// TIA Portal V16 program export: 1 tag tables, 0 data types, 1 data blocks, 5 code blocks (in call order from the OBs), 0 instance data blocks

VAR_GLOBAL   // PLC tag table "Default tag table"
   inp_1_tia_da_degisti AT %M0.0 : Bool;
   out_1_degistirildi AT %M0.1 : Bool;
END_VAR

DATA_BLOCK "Data_block_1"   // DB1
{ S7_Optimized_Access := 'TRUE' }
VERSION : 0.1
// stored: AutoNumber true, DBAccessibleFromOPCUA true, IsOnlyStoredInLoadMemory false, IsRetainMemResEnabled false, IsWriteProtectedInAS false, MemoryReserve 100
   VAR
      ex : Bool;
      ex_1 : Bool;
      ex_2 : Bool;
      ex_3 : Bool;
      ex_4 : Bool;
      ex_5 : Bool;
      ex_6 : Bool;
      ex_7 : Bool;
      ex_8 : Bool;
      ex_9 : Bool;
      new : Bool;
      new_1 : Bool;
      new_2 : Bool;
   END_VAR
BEGIN
END_DATA_BLOCK

ORGANIZATION_BLOCK "Main"   // OB1, LAD, ProgramCycle
TITLE = "Main Program Sweep (Cycle)"
{ S7_Optimized_Access := 'TRUE' }
VERSION : 0.1
// stored: AutoNumber true, IsIECCheckEnabled false, SetENOAutomatically false
   VAR_INPUT
      Initial_Call : Bool;   // Initial call of this OB
      Remanence : Bool;   // =True, if remanent data are available
   END_VAR
   VAR_TEMP
      deneme_123 : Bool;
      deneme_2 : Bool;
   END_VAR
BEGIN

REGION Network 1: yorum111
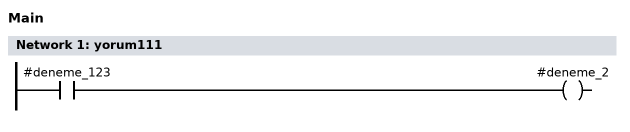
   RUNG wire#powerrail
      Contact( #deneme_123 )
      Coil( #deneme_2 )
   END_RUNG
   // the same network as SCL:
   #deneme_2 := #deneme_123;
END_REGION
END_ORGANIZATION_BLOCK

FUNCTION "Block_1" : Void   // FC2, LAD
{ S7_Optimized_Access := 'TRUE' }
VERSION : 0.1
// stored: AutoNumber true, IsIECCheckEnabled false, SetENOAutomatically false, UDAEnableTagReadback false
BEGIN
END_FUNCTION

FUNCTION "analog_output_scale" : Void   // FC1, LAD
{ S7_Optimized_Access := 'TRUE' }
VERSION : 0.1
// stored: AutoNumber true, IsIECCheckEnabled false, SetENOAutomatically false, UDAEnableTagReadback false
BEGIN

REGION Network 1
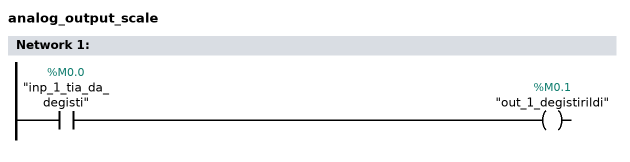
   RUNG wire#powerrail
      Contact( "inp_1_tia_da_degisti" )
      Coil( "out_1_degistirildi" )
   END_RUNG
   // the same network as SCL:
   "out_1_degistirildi" := "inp_1_tia_da_degisti";
END_REGION
END_FUNCTION

FUNCTION_BLOCK "FB548.Divert.Sorter.Chute"   // FB542, LAD
{ S7_Optimized_Access := 'TRUE' }
VERSION : 0.1
// stored: AutoNumber false, IsIECCheckEnabled false, IsRetainMemResEnabled false, MemoryReserve 100, SetENOAutomatically false, UDAEnableTagReadback false
   VAR_INPUT
      Acil_Yok : Bool;
      Sorter_Calisiyor : Bool;
      Sağ_Chute_Sorted_Sensoru : Bool;
      Sol_Chute_Sorted_Sensoru : Bool;
      "Sağ_Chute_Aktif / Pasif" : Bool;   // 1 = Aktif , 0 = Pasif
      "Sol_Chute_Aktif / Pasif" : Bool;   // 1 = Aktif , 0 = Pasif
      Chute_Rulo_Hatası : Bool;
      Divert_Sürücü_Hatası : Bool;
      Pozisyon_Olcme_Aktif : Bool;
      Sağ_Çıkış_Target { ExternalAccessible := 'False'; ExternalVisible := 'False'; ExternalWritable := 'False'} : Int;
      Sol_Çıkış_Target { ExternalAccessible := 'False'; ExternalVisible := 'False'; ExternalWritable := 'False'} : Int;
      CN_NO : Int;
      "Aktüel Encoder Değeri" : LReal;
      Birinci_Divert_Min : LReal;
      Birinci_Divert_Max : LReal;
      İkinci_Divert_Min : LReal;
      İkinci_Divert_Max : LReal;
      Max_Kutu_Adedi { ExternalAccessible := 'False'; ExternalVisible := 'False'; ExternalWritable := 'False'} : Int;
   END_VAR
   VAR_OUTPUT
      "1_sol_Divert_Çalıştır" : Bool;
      "2_sol_Divert_Çalıştır" : Bool;
      "1_sağ_Divert_Çalıştır" : Bool;
      "2_sağ_Divert_Çalıştır" : Bool;
      "Sort Hatası" : Bool;
   END_VAR
   VAR
      Sort_Aktif_AUX : Array[1..10] of Bool;
      Sort_Aktif_PTrig : Array[1..10] of Bool;
      TOF_TIME : Array[1..10] of TOF_TIME;
      TON_TIME { S7_SetPoint := 'True'} : Array[1..10] of TON_TIME;
      Sort_Aktif1 : Bool;
      Sort_Aktif2 : Bool;
      Sort_Aktif1_Sağ : Bool;
      Sort_Aktif2_Sağ : Bool;
      Sağ_Sort_Pasif : Bool;
      Sol_Sort_Pasif : Bool;
      Ikinci_Servo_Baslama : Time;
      Divert_Durdur : Bool;
      Sort_Aktif_1 { ExternalAccessible := 'False'; ExternalVisible := 'False'; ExternalWritable := 'False'} : Array[1..10] of Bool;
      Sort_Aktif_2 { ExternalAccessible := 'False'; ExternalVisible := 'False'; ExternalWritable := 'False'} : Array[1..10] of Bool;
      Sort_Aktif_1_Sağ : Array[1..10] of Bool;
      Sort_Aktif_2_Sağ : Array[1..10] of Bool;
      Sort_Ilk_Pozisyon { ExternalAccessible := 'False'; ExternalVisible := 'False'; ExternalWritable := 'False'} : Array[1..10] of LReal;
      Sort_Ön_Pozisyon { ExternalAccessible := 'False'; ExternalVisible := 'False'; ExternalWritable := 'False'} : Array[1..10] of LReal;
      Sort_Aktif_Boy { ExternalAccessible := 'False'; ExternalVisible := 'False'; ExternalWritable := 'False'} : Array[1..10] of LReal;
      SortKutuNo : Int;
   END_VAR
   VAR_TEMP
      "On/Off" : Bool;
      j : Int;
      Ekstra_Uzunluk : LReal;
   END_VAR
   VAR_TEMP   // added for the SCL form of the ladder/FBD networks
      _w1 : Bool;
      _w2 : Bool;
      _w3 : Bool;
      _w4 : Bool;
   END_VAR
BEGIN

REGION Network 1: On / Off
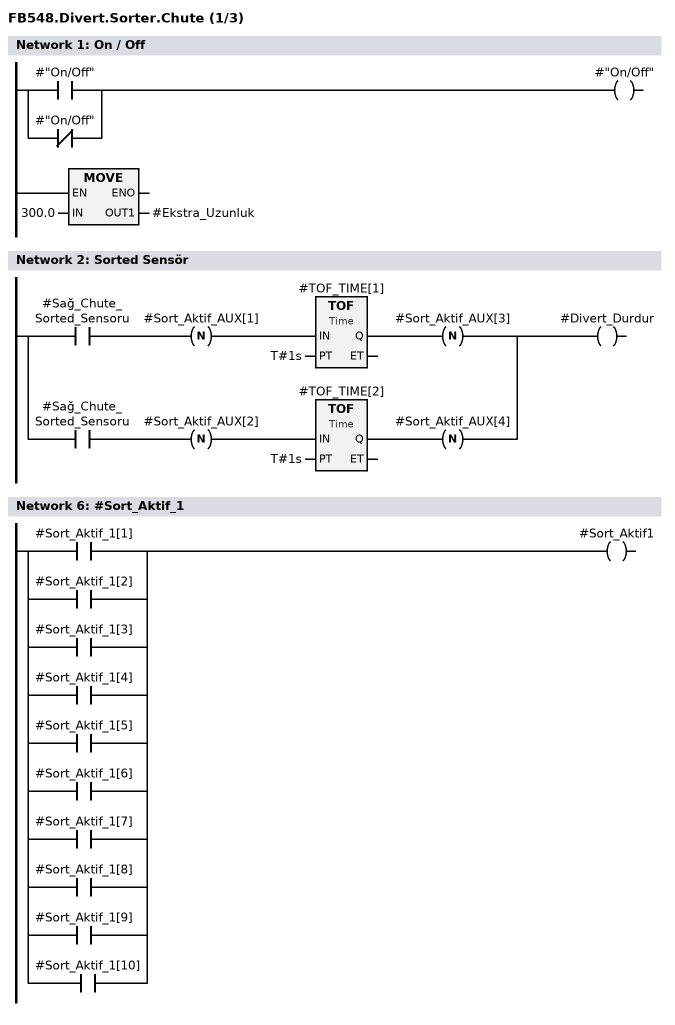
   RUNG wire#powerrail
      Contact( #"On/Off" )
      wire#w1
      Coil( #"On/Off" )
   END_RUNG
   RUNG wire#powerrail
      I_Contact( #"On/Off" )
   END_RUNG wire#w1
   RUNG wire#powerrail
      Move(in := 300.0, out1 => #Ekstra_Uzunluk)
   END_RUNG
   // the same network as SCL:
   #"On/Off" := #"On/Off" OR NOT #"On/Off";
   #Ekstra_Uzunluk := 300.0;
END_REGION

REGION Network 2: Sorted Sensör
   RUNG wire#powerrail
      Contact( #Sağ_Chute_Sorted_Sensoru )
      N_Trig( #Sort_Aktif_AUX[1] )
      { S7_Templates := "time_type := Time" } #TOF_TIME[1].TOF(pt := T#1s, et =>)
      N_Trig( #Sort_Aktif_AUX[3] )
      wire#w1
      Coil( #Divert_Durdur )
   END_RUNG
   RUNG wire#powerrail
      Contact( #Sağ_Chute_Sorted_Sensoru )
      N_Trig( #Sort_Aktif_AUX[2] )
      { S7_Templates := "time_type := Time" } #TOF_TIME[2].TOF(pt := T#1s, et =>)
      N_Trig( #Sort_Aktif_AUX[4] )
   END_RUNG wire#w1
   // the same network as SCL:
   #_w1 := NOT #Sağ_Chute_Sorted_Sensoru AND #Sort_Aktif_AUX[1];   // falling edge
   #Sort_Aktif_AUX[1] := #Sağ_Chute_Sorted_Sensoru;
   #TOF_TIME[1].TOF(IN := #_w1, PT := T#1s);
   #_w2 := NOT #TOF_TIME[1].Q AND #Sort_Aktif_AUX[3];   // falling edge
   #Sort_Aktif_AUX[3] := #TOF_TIME[1].Q;
   #_w3 := NOT #Sağ_Chute_Sorted_Sensoru AND #Sort_Aktif_AUX[2];   // falling edge
   #Sort_Aktif_AUX[2] := #Sağ_Chute_Sorted_Sensoru;
   #TOF_TIME[2].TOF(IN := #_w3, PT := T#1s);
   #_w4 := NOT #TOF_TIME[2].Q AND #Sort_Aktif_AUX[4];   // falling edge
   #Sort_Aktif_AUX[4] := #TOF_TIME[2].Q;
   #Divert_Durdur := #_w2 OR #_w4;
END_REGION

REGION Network 3 (SCL): Kutu Ön Arka Pozisyon Hesap
   // IF #Sensör.Sensor_N_Trig THEN
   //     #Sort_Ilk_Pozisyon["DB530_Kutu".CN_NO_Anlık_Kutu_Sayısı[#CN_NO]] := #"Aktüel Encoder Değeri";
   // END_IF;
   // FOR #j := 1 TO #Max_Kutu_Adedi BY 1 DO
   //     IF "DB530_Kutu".CN_NO[#CN_NO].Kutu_No[#j].VARMI = TRUE THEN
   //         #Sort_Ön_Pozisyon[#j] := #"Aktüel Encoder Değeri" - #Sort_Ilk_Pozisyon[#j];
   //     END_IF;
   // END_FOR;
END_REGION

REGION Network 4 (SCL): Sol Sort Aktif Kararı
   IF #Pozisyon_Olcme_Aktif = 0
       // AND #Sorter_Calisiyor = TRUE
       // AND #"Sol_Chute_Aktif / Pasif"
   THEN
       FOR #j := 1 TO #Max_Kutu_Adedi BY 1 DO
           IF "DB530_Kutu".CN_NO[#CN_NO].Kutu_No[#j].VARMI THEN

               IF #"Sol_Chute_Aktif / Pasif" = 1
                   AND #Chute_Rulo_Hatası = 0
                   AND #Divert_Sürücü_Hatası = 0
                   // AND #Sol_Sort_Pasif = 0
                   AND #Acil_Yok = 1
                   AND "DB530_Kutu".CN_NO[#CN_NO].Kutu_No[#j].Posizyon >= #Birinci_Divert_Min
                   AND "DB530_Kutu".CN_NO[#CN_NO].Kutu_No[#j].Posizyon <= #Birinci_Divert_Min + "DB530_Kutu".CN_NO[#CN_NO].Kutu_No[#j].Uzunluk + #Ekstra_Uzunluk
                   AND "DB530_Kutu".CN_NO[#CN_NO].Kutu_No[#j].Target = #Sol_Çıkış_Target
                   // AND "DB530_Kutu".CN_NO[#CN_NO].Kutu_No[#j].Sort_Aktifleştirildi = FALSE
               THEN
                   #Sort_Aktif_1[#j] := TRUE;
               ELSE

                   IF #j< #Max_Kutu_Adedi THEN
                       IF ("DB530_Kutu".CN_NO[#CN_NO].Kutu_No[#j + 1].VARMI AND "DB530_Kutu".CN_NO[#CN_NO].Kutu_No[#j + 1].Target = #Sol_Çıkış_Target)
                           OR ("DB530_Kutu".CN_NO[#CN_NO].Kutu_No[#j].VARMI AND "DB530_Kutu".CN_NO[#CN_NO].Kutu_No[#j].Target = #Sol_Çıkış_Target) THEN

                           #Sort_Aktif_1[#j] := TRUE;

                       ELSE
                           #Sort_Aktif_1[#j] := FALSE;
                       END_IF;

                   END_IF;

               END_IF;

               IF #"Sol_Chute_Aktif / Pasif" = 1
                   AND #Chute_Rulo_Hatası = 0
                   AND #Divert_Sürücü_Hatası = 0
                   // AND #Sol_Sort_Pasif = 0
                   AND #Acil_Yok = 1
                   AND "DB530_Kutu".CN_NO[#CN_NO].Kutu_No[#j].Posizyon >= #İkinci_Divert_Min
                   AND "DB530_Kutu".CN_NO[#CN_NO].Kutu_No[#j].Posizyon <= #İkinci_Divert_Min + "DB530_Kutu".CN_NO[#CN_NO].Kutu_No[#j].Uzunluk + #Ekstra_Uzunluk
                   AND "DB530_Kutu".CN_NO[#CN_NO].Kutu_No[#j].Target = #Sol_Çıkış_Target
                   // AND "DB530_Kutu".CN_NO[#CN_NO].Kutu_No[#j].Sort_Aktifleştirildi = FALSE
               THEN
                   #Sort_Aktif_2[#j] := TRUE;
               ELSE
                   IF #j < #Max_Kutu_Adedi THEN
                       IF ("DB530_Kutu".CN_NO[#CN_NO].Kutu_No[#j + 1].VARMI AND "DB530_Kutu".CN_NO[#CN_NO].Kutu_No[#j + 1].Target = #Sol_Çıkış_Target )
                           OR ("DB530_Kutu".CN_NO[#CN_NO].Kutu_No[#j].VARMI AND "DB530_Kutu".CN_NO[#CN_NO].Kutu_No[#j].Target = #Sol_Çıkış_Target) THEN

                           #Sort_Aktif_2[#j] := TRUE;

                       ELSE
                           #Sort_Aktif_2[#j] := FALSE;
                       END_IF;

                   END_IF;
               END_IF;

               // IF "DB530_Kutu".CN_NO[#CN_NO].Kutu_No[#j].Posizyon > #İkinci_Divert_Max + "DB530_Kutu".CN_NO[#CN_NO].Kutu_No[#j].Uzunluk THEN
               //     "DB530_Kutu".CN_NO[#CN_NO].Kutu_No[#j].Sort_Aktifleştirildi := true;
               // END_IF;

               ///////////SortStatus//SolTaraf
               IF "DB530_Kutu".CN_NO[#CN_NO].Kutu_No[#j].Target = #Sol_Çıkış_Target // Sol Çıkış Statüleri
                   // AND "DB530_Kutu".CN_NO[#CN_NO].Kutu_No[#j].VARMI = True
                   AND ("DB530_Kutu".CN_NO[#CN_NO].Kutu_No[#j].Posizyon >= #Birinci_Divert_Min OR "DB530_Kutu".CN_NO[#CN_NO].Kutu_No[#j].Posizyon >= #İkinci_Divert_Min)
                   // AND "DB530_Kutu".CN_NO[#CN_NO].Kutu_No[#j].Sort_Aktifleştirildi = 0
                   // AND (#"Sol_Chute_Aktif / Pasif" = 0 OR #Divert_Sürücü_Hatası = 1 OR #Chute_Rulo_Hatası = 1)
               THEN
                   IF #"Sol_Chute_Aktif / Pasif" = 0 OR #Acil_Yok = 0 THEN
                       "DB530_Kutu".CN_NO[#CN_NO].Kutu_No[#j].Sort_Statu := 1;
                       // "DB530_Kutu".CN_NO[#CN_NO].Kutu_No[#j].Sort_Aktifleştirildi := 1;
                   ELSIF #Divert_Sürücü_Hatası = 1 THEN
                       "DB530_Kutu".CN_NO[#CN_NO].Kutu_No[#j].Sort_Statu := 2;
                       // "DB530_Kutu".CN_NO[#CN_NO].Kutu_No[#j].Sort_Aktifleştirildi := 1;
                   ELSIF #Chute_Rulo_Hatası = 1 THEN
                       "DB530_Kutu".CN_NO[#CN_NO].Kutu_No[#j].Sort_Statu := 3;
                       // "DB530_Kutu".CN_NO[#CN_NO].Kutu_No[#j].Sort_Aktifleştirildi := 1;
                   ELSIF (#Sort_Aktif_1[#j] = 1 OR #Sort_Aktif_2[#j] = 1) THEN
                       "DB530_Kutu".CN_NO[#CN_NO].Kutu_No[#j].Sort_Statu := 10;
                       "DB530_Kutu".CN_NO[#CN_NO].Kutu_No[#j].Sort_Aktifleştirildi := 1;
                       "DB542.Chute.Kontrol".CN_NO[#CN_NO].Sort_UID_Kutu_No[#j] := "DB530_Kutu".CN_NO[#CN_NO].Kutu_No[#j].UniqueID;
                   END_IF;
               END_IF;
           END_IF;
           IF "DB530_Kutu".CN_NO[#CN_NO].Kutu_No[1].VARMI = 0 THEN
               #Sort_Aktif_1[#j] := FALSE;
               #Sort_Aktif_2[#j] := FALSE;
           END_IF;
       END_FOR;
   END_IF;
END_REGION

REGION Network 5 (SCL): Sağ Sort Aktif Kararı
   IF #Pozisyon_Olcme_Aktif = 0
       // AND #Sorter_Calisiyor = TRUE
       // AND #"Sağ_Chute_Aktif / Pasif"
   THEN

       FOR #j := 1 TO #Max_Kutu_Adedi BY 1 DO
           IF "DB530_Kutu".CN_NO[#CN_NO].Kutu_No[#j].VARMI THEN


               IF #"Sağ_Chute_Aktif / Pasif" = 1
                   AND #Chute_Rulo_Hatası = 0
                   AND #Divert_Sürücü_Hatası = 0
                   // AND #Sağ_Sort_Pasif = 0
                   AND #Acil_Yok = 1
                   AND "DB530_Kutu".CN_NO[#CN_NO].Kutu_No[#j].Posizyon >= #Birinci_Divert_Min
                   AND "DB530_Kutu".CN_NO[#CN_NO].Kutu_No[#j].Posizyon <= #Birinci_Divert_Min + "DB530_Kutu".CN_NO[#CN_NO].Kutu_No[#j].Uzunluk + #Ekstra_Uzunluk
                   AND "DB530_Kutu".CN_NO[#CN_NO].Kutu_No[#j].Target = #Sağ_Çıkış_Target
                   // AND "DB530_Kutu".CN_NO[#CN_NO].Kutu_No[#j].Sort_Aktifleştirildi = FALSE
               THEN
                   #Sort_Aktif_1_Sağ[#j] := TRUE;
               ELSE
                   IF #j < #Max_Kutu_Adedi THEN
                       IF ("DB530_Kutu".CN_NO[#CN_NO].Kutu_No[#j + 1].VARMI AND "DB530_Kutu".CN_NO[#CN_NO].Kutu_No[#j + 1].Target = #Sağ_Çıkış_Target)
                           OR ("DB530_Kutu".CN_NO[#CN_NO].Kutu_No[#j].VARMI AND "DB530_Kutu".CN_NO[#CN_NO].Kutu_No[#j].Target = #Sağ_Çıkış_Target) THEN

                           #Sort_Aktif_1_Sağ[#j] := TRUE;

                       ELSE
                           #Sort_Aktif_1_Sağ[#j] := FALSE;
                       END_IF;

                   END_IF;

               END_IF;

               IF #"Sağ_Chute_Aktif / Pasif" = 1
                   AND #Chute_Rulo_Hatası = 0
                   AND #Divert_Sürücü_Hatası = 0
                   // AND #Sağ_Sort_Pasif = 0
                   AND #Acil_Yok = 1
                   AND "DB530_Kutu".CN_NO[#CN_NO].Kutu_No[#j].Posizyon >= #İkinci_Divert_Min
                   AND "DB530_Kutu".CN_NO[#CN_NO].Kutu_No[#j].Posizyon <= #İkinci_Divert_Min + "DB530_Kutu".CN_NO[#CN_NO].Kutu_No[#j].Uzunluk + #Ekstra_Uzunluk
                   AND "DB530_Kutu".CN_NO[#CN_NO].Kutu_No[#j].Target = #Sağ_Çıkış_Target
                   // AND "DB530_Kutu".CN_NO[#CN_NO].Kutu_No[#j].Sort_Aktifleştirildi = FALSE
               THEN
                   #Sort_Aktif_2_Sağ[#j] := TRUE;
               ELSE
                   IF #j < #Max_Kutu_Adedi THEN
                       IF ("DB530_Kutu".CN_NO[#CN_NO].Kutu_No[#j + 1].VARMI AND "DB530_Kutu".CN_NO[#CN_NO].Kutu_No[#j + 1].Target = #Sağ_Çıkış_Target )
                           OR ("DB530_Kutu".CN_NO[#CN_NO].Kutu_No[#j].VARMI AND "DB530_Kutu".CN_NO[#CN_NO].Kutu_No[#j].Target = #Sağ_Çıkış_Target) THEN

                           #Sort_Aktif_2_Sağ[#j] := TRUE;

                       ELSE
                           #Sort_Aktif_2_Sağ[#j] := FALSE;
                       END_IF;

                   END_IF;

               END_IF;

               // IF "DB530_Kutu".CN_NO[#CN_NO].Kutu_No[#j].Posizyon > #İkinci_Divert_Max + "DB530_Kutu".CN_NO[#CN_NO].Kutu_No[#j].Uzunluk THEN
               //     "DB530_Kutu".CN_NO[#CN_NO].Kutu_No[#j].Sort_Aktifleştirildi := true;
               // END_IF;

               ///////////SortStatus//SağTaraf
               IF "DB530_Kutu".CN_NO[#CN_NO].Kutu_No[#j].Target = #Sağ_Çıkış_Target // Sağ Çıkış Statüleri
                   // AND "DB530_Kutu".CN_NO[#CN_NO].Kutu_No[#j].VARMI = True
                   AND ("DB530_Kutu".CN_NO[#CN_NO].Kutu_No[#j].Posizyon >= #Birinci_Divert_Min OR "DB530_Kutu".CN_NO[#CN_NO].Kutu_No[#j].Posizyon >= #İkinci_Divert_Min)
                   // AND "DB530_Kutu".CN_NO[#CN_NO].Kutu_No[#j].Sort_Aktifleştirildi = 0
                   // AND (#"Sağ_Chute_Aktif / Pasif" = 0 OR #Divert_Sürücü_Hatası = 1 OR #Chute_Rulo_Hatası = 1)
               THEN
                   IF #"Sağ_Chute_Aktif / Pasif" = 0 OR #Acil_Yok = 0 THEN
                       "DB530_Kutu".CN_NO[#CN_NO].Kutu_No[#j].Sort_Statu := 1;
                       // "DB530_Kutu".CN_NO[#CN_NO].Kutu_No[#j].Sort_Aktifleştirildi := 1;
                   ELSIF #Divert_Sürücü_Hatası = 1 THEN
                       "DB530_Kutu".CN_NO[#CN_NO].Kutu_No[#j].Sort_Statu := 2;
                       // "DB530_Kutu".CN_NO[#CN_NO].Kutu_No[#j].Sort_Aktifleştirildi := 1;
                   ELSIF #Chute_Rulo_Hatası = 1 THEN
                       "DB530_Kutu".CN_NO[#CN_NO].Kutu_No[#j].Sort_Statu := 3;
                       // "DB530_Kutu".CN_NO[#CN_NO].Kutu_No[#j].Sort_Aktifleştirildi := 1;
                   ELSIF (#Sort_Aktif_1_Sağ[#j] = 1 OR #Sort_Aktif_2_Sağ[#j] = 1) THEN
                       "DB530_Kutu".CN_NO[#CN_NO].Kutu_No[#j].Sort_Statu := 10;
                       "DB530_Kutu".CN_NO[#CN_NO].Kutu_No[#j].Sort_Aktifleştirildi := 1;
                       "DB542.Chute.Kontrol".CN_NO[#CN_NO].Sort_UID_Kutu_No[#j] := "DB530_Kutu".CN_NO[#CN_NO].Kutu_No[#j].UniqueID;
                   END_IF;
               END_IF;
           END_IF;
           IF "DB530_Kutu".CN_NO[#CN_NO].Kutu_No[1].VARMI = 0 THEN
               #Sort_Aktif_1_Sağ[#j] := FALSE;
               #Sort_Aktif_2_Sağ[#j] := FALSE;
           END_IF;
       END_FOR;
   END_IF;
END_REGION

REGION Network 6: #Sort_Aktif_1
   RUNG wire#powerrail
      Contact( #Sort_Aktif_1[1] )
      wire#w1
      Coil( #Sort_Aktif1 )
   END_RUNG
   RUNG wire#powerrail
      Contact( #Sort_Aktif_1[2] )
   END_RUNG wire#w1
   RUNG wire#powerrail
      Contact( #Sort_Aktif_1[3] )
   END_RUNG wire#w1
   RUNG wire#powerrail
      Contact( #Sort_Aktif_1[4] )
   END_RUNG wire#w1
   RUNG wire#powerrail
      Contact( #Sort_Aktif_1[5] )
   END_RUNG wire#w1
   RUNG wire#powerrail
      Contact( #Sort_Aktif_1[6] )
   END_RUNG wire#w1
   RUNG wire#powerrail
      Contact( #Sort_Aktif_1[7] )
   END_RUNG wire#w1
   RUNG wire#powerrail
      Contact( #Sort_Aktif_1[8] )
   END_RUNG wire#w1
   RUNG wire#powerrail
      Contact( #Sort_Aktif_1[9] )
   END_RUNG wire#w1
   RUNG wire#powerrail
      Contact( #Sort_Aktif_1[10] )
   END_RUNG wire#w1
   // the same network as SCL:
   #Sort_Aktif1 := #Sort_Aktif_1[1] OR #Sort_Aktif_1[2] OR #Sort_Aktif_1[3] OR #Sort_Aktif_1[4] OR #Sort_Aktif_1[5] OR #Sort_Aktif_1[6] OR #Sort_Aktif_1[7] OR #Sort_Aktif_1[8] OR #Sort_Aktif_1[9] OR #Sort_Aktif_1[10];
END_REGION

REGION Network 7: #Sort_Aktif_2
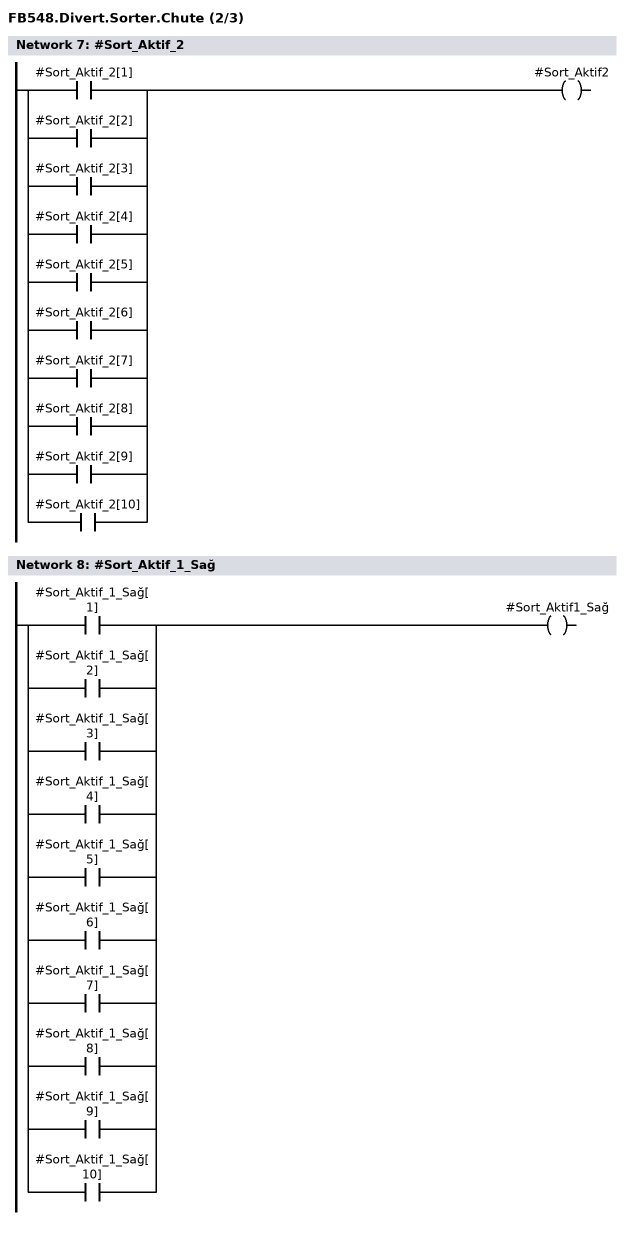
   RUNG wire#powerrail
      Contact( #Sort_Aktif_2[1] )
      wire#w1
      Coil( #Sort_Aktif2 )
   END_RUNG
   RUNG wire#powerrail
      Contact( #Sort_Aktif_2[2] )
   END_RUNG wire#w1
   RUNG wire#powerrail
      Contact( #Sort_Aktif_2[3] )
   END_RUNG wire#w1
   RUNG wire#powerrail
      Contact( #Sort_Aktif_2[4] )
   END_RUNG wire#w1
   RUNG wire#powerrail
      Contact( #Sort_Aktif_2[5] )
   END_RUNG wire#w1
   RUNG wire#powerrail
      Contact( #Sort_Aktif_2[6] )
   END_RUNG wire#w1
   RUNG wire#powerrail
      Contact( #Sort_Aktif_2[7] )
   END_RUNG wire#w1
   RUNG wire#powerrail
      Contact( #Sort_Aktif_2[8] )
   END_RUNG wire#w1
   RUNG wire#powerrail
      Contact( #Sort_Aktif_2[9] )
   END_RUNG wire#w1
   RUNG wire#powerrail
      Contact( #Sort_Aktif_2[10] )
   END_RUNG wire#w1
   // the same network as SCL:
   #Sort_Aktif2 := #Sort_Aktif_2[1] OR #Sort_Aktif_2[2] OR #Sort_Aktif_2[3] OR #Sort_Aktif_2[4] OR #Sort_Aktif_2[5] OR #Sort_Aktif_2[6] OR #Sort_Aktif_2[7] OR #Sort_Aktif_2[8] OR #Sort_Aktif_2[9] OR #Sort_Aktif_2[10];
END_REGION

REGION Network 8: #Sort_Aktif_1_Sağ
   RUNG wire#powerrail
      Contact( #Sort_Aktif_1_Sağ[1] )
      wire#w1
      Coil( #Sort_Aktif1_Sağ )
   END_RUNG
   RUNG wire#powerrail
      Contact( #Sort_Aktif_1_Sağ[2] )
   END_RUNG wire#w1
   RUNG wire#powerrail
      Contact( #Sort_Aktif_1_Sağ[3] )
   END_RUNG wire#w1
   RUNG wire#powerrail
      Contact( #Sort_Aktif_1_Sağ[4] )
   END_RUNG wire#w1
   RUNG wire#powerrail
      Contact( #Sort_Aktif_1_Sağ[5] )
   END_RUNG wire#w1
   RUNG wire#powerrail
      Contact( #Sort_Aktif_1_Sağ[6] )
   END_RUNG wire#w1
   RUNG wire#powerrail
      Contact( #Sort_Aktif_1_Sağ[7] )
   END_RUNG wire#w1
   RUNG wire#powerrail
      Contact( #Sort_Aktif_1_Sağ[8] )
   END_RUNG wire#w1
   RUNG wire#powerrail
      Contact( #Sort_Aktif_1_Sağ[9] )
   END_RUNG wire#w1
   RUNG wire#powerrail
      Contact( #Sort_Aktif_1_Sağ[10] )
   END_RUNG wire#w1
   // the same network as SCL:
   #Sort_Aktif1_Sağ := #Sort_Aktif_1_Sağ[1] OR #Sort_Aktif_1_Sağ[2] OR #Sort_Aktif_1_Sağ[3] OR #Sort_Aktif_1_Sağ[4] OR #Sort_Aktif_1_Sağ[5] OR #Sort_Aktif_1_Sağ[6] OR #Sort_Aktif_1_Sağ[7] OR #Sort_Aktif_1_Sağ[8] OR #Sort_Aktif_1_Sağ[9] OR #Sort_Aktif_1_Sağ[10];
END_REGION

REGION Network 9: #Sort_Aktif_2_Sağ
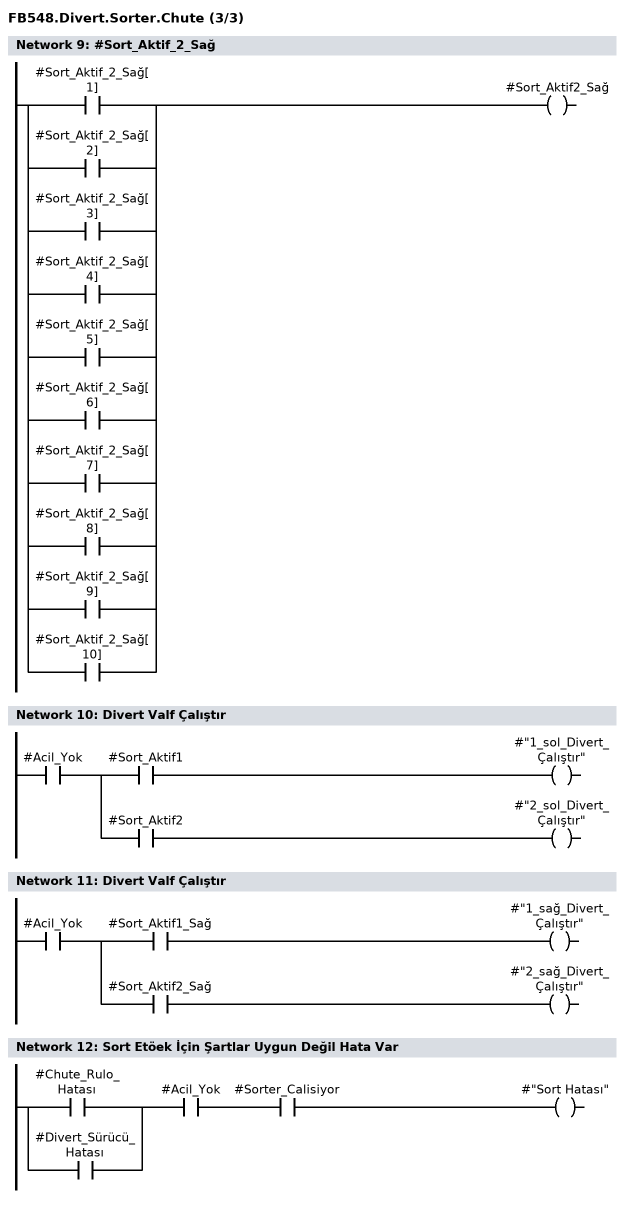
   RUNG wire#powerrail
      Contact( #Sort_Aktif_2_Sağ[1] )
      wire#w1
      Coil( #Sort_Aktif2_Sağ )
   END_RUNG
   RUNG wire#powerrail
      Contact( #Sort_Aktif_2_Sağ[2] )
   END_RUNG wire#w1
   RUNG wire#powerrail
      Contact( #Sort_Aktif_2_Sağ[3] )
   END_RUNG wire#w1
   RUNG wire#powerrail
      Contact( #Sort_Aktif_2_Sağ[4] )
   END_RUNG wire#w1
   RUNG wire#powerrail
      Contact( #Sort_Aktif_2_Sağ[5] )
   END_RUNG wire#w1
   RUNG wire#powerrail
      Contact( #Sort_Aktif_2_Sağ[6] )
   END_RUNG wire#w1
   RUNG wire#powerrail
      Contact( #Sort_Aktif_2_Sağ[7] )
   END_RUNG wire#w1
   RUNG wire#powerrail
      Contact( #Sort_Aktif_2_Sağ[8] )
   END_RUNG wire#w1
   RUNG wire#powerrail
      Contact( #Sort_Aktif_2_Sağ[9] )
   END_RUNG wire#w1
   RUNG wire#powerrail
      Contact( #Sort_Aktif_2_Sağ[10] )
   END_RUNG wire#w1
   // the same network as SCL:
   #Sort_Aktif2_Sağ := #Sort_Aktif_2_Sağ[1] OR #Sort_Aktif_2_Sağ[2] OR #Sort_Aktif_2_Sağ[3] OR #Sort_Aktif_2_Sağ[4] OR #Sort_Aktif_2_Sağ[5] OR #Sort_Aktif_2_Sağ[6] OR #Sort_Aktif_2_Sağ[7] OR #Sort_Aktif_2_Sağ[8] OR #Sort_Aktif_2_Sağ[9] OR #Sort_Aktif_2_Sağ[10];
END_REGION

REGION Network 10: Divert Valf Çalıştır
   RUNG wire#powerrail
      Contact( #Acil_Yok )
      wire#w1
      Contact( #Sort_Aktif1 )
      Coil( #"1_sol_Divert_Çalıştır" )
   END_RUNG
   RUNG wire#w1
      Contact( #Sort_Aktif2 )
      Coil( #"2_sol_Divert_Çalıştır" )
   END_RUNG
   // the same network as SCL:
   #"1_sol_Divert_Çalıştır" := #Acil_Yok AND #Sort_Aktif1;
   #"2_sol_Divert_Çalıştır" := #Acil_Yok AND #Sort_Aktif2;
END_REGION

REGION Network 11: Divert Valf Çalıştır
   RUNG wire#powerrail
      Contact( #Acil_Yok )
      wire#w1
      Contact( #Sort_Aktif1_Sağ )
      Coil( #"1_sağ_Divert_Çalıştır" )
   END_RUNG
   RUNG wire#w1
      Contact( #Sort_Aktif2_Sağ )
      Coil( #"2_sağ_Divert_Çalıştır" )
   END_RUNG
   // the same network as SCL:
   #"1_sağ_Divert_Çalıştır" := #Acil_Yok AND #Sort_Aktif1_Sağ;
   #"2_sağ_Divert_Çalıştır" := #Acil_Yok AND #Sort_Aktif2_Sağ;
END_REGION

REGION Network 12: Sort Etöek İçin Şartlar Uygun Değil Hata Var
   RUNG wire#powerrail
      Contact( #Chute_Rulo_Hatası )
      wire#w1
      Contact( #Acil_Yok )
      Contact( #Sorter_Calisiyor )
      Coil( #"Sort Hatası" )
   END_RUNG
   RUNG wire#powerrail
      Contact( #Divert_Sürücü_Hatası )
   END_RUNG wire#w1
   // the same network as SCL:
   #"Sort Hatası" := (#Chute_Rulo_Hatası OR #Divert_Sürücü_Hatası) AND #Acil_Yok AND #Sorter_Calisiyor;
END_REGION
END_FUNCTION_BLOCK

FUNCTION_BLOCK "FB_ChuteControl"   // FB4, LAD
{ S7_Optimized_Access := 'TRUE' }
VERSION : 0.1
// stored: AutoNumber true, IsIECCheckEnabled false, IsRetainMemResEnabled false, MemoryReserve 100, SetENOAutomatically false, UDAEnableTagReadback false
   VAR_INPUT
      Acil_OK : Bool;
      Otomatik : Bool;
      Hata_Reset : Bool;
   END_VAR
   VAR
      Yanaştırma : "FB549.Divert.Sorter.Basing";
      "FB548.Divert.Sorter.Chute_CN1_Divert1" { S7_SetPoint := 'True'} : "FB548.Divert.Sorter.Chute";
      "FB548.Divert.Sorter.Chute_CN2_Divert2" { S7_SetPoint := 'True'} : "FB548.Divert.Sorter.Chute";
      "FB548.Divert.Sorter.Chute_CN3_Divert3" { S7_SetPoint := 'True'} : "FB548.Divert.Sorter.Chute";
      "FB548.Divert.Sorter.Chute_CN4_Divert4" { S7_SetPoint := 'True'} : "FB548.Divert.Sorter.Chute";
      "FB548.Divert.Sorter.Chute_CN5_Divert5" { S7_SetPoint := 'True'} : "FB548.Divert.Sorter.Chute";
   END_VAR
   VAR_TEMP
      i : Int;
      j : Int;
   END_VAR
   VAR_TEMP   // added for the SCL form of the ladder/FBD networks
      _w1 : Bool;
   END_VAR
BEGIN

REGION Network 1: CN2 POS1065 Divert1
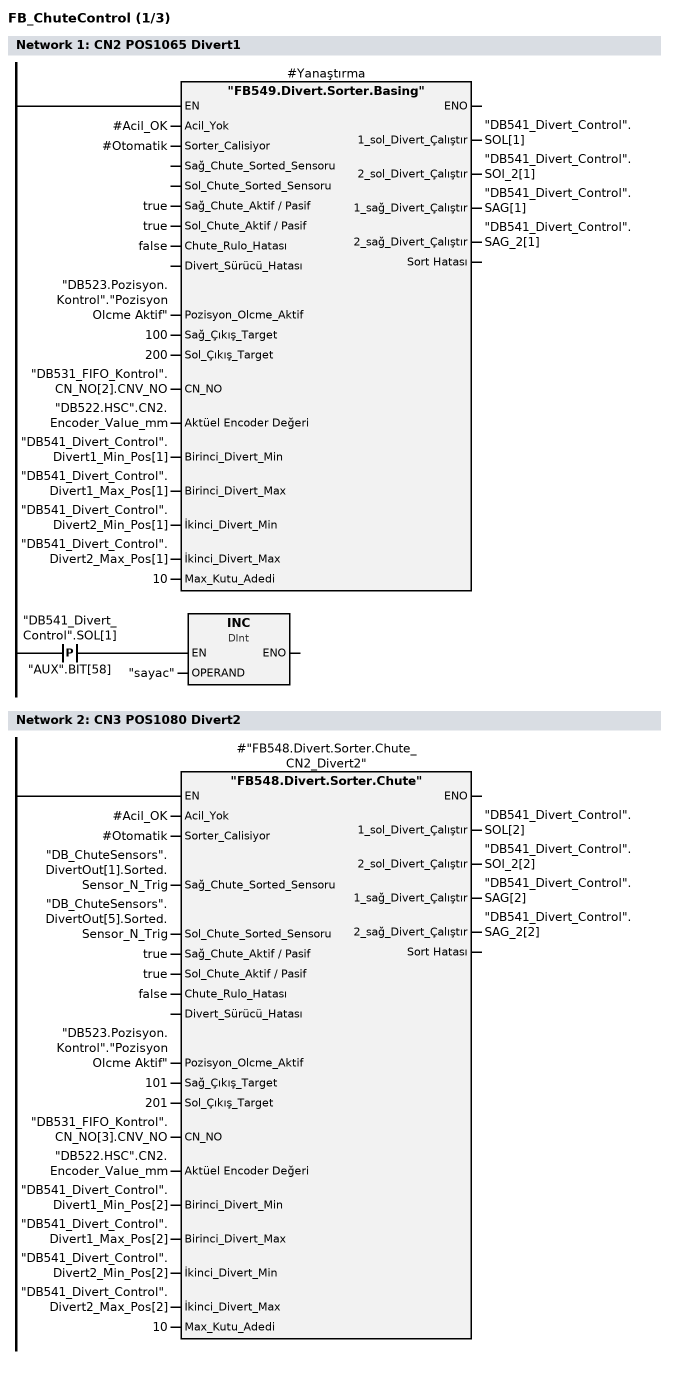
   RUNG wire#powerrail
      #Yanaştırma(Acil_Yok := #Acil_OK, Sorter_Calisiyor := #Otomatik, Sağ_Chute_Sorted_Sensoru :=, Sol_Chute_Sorted_Sensoru :=, "Sağ_Chute_Aktif / Pasif" := true, "Sol_Chute_Aktif / Pasif" := true, Chute_Rulo_Hatası := false, Divert_Sürücü_Hatası :=, Pozisyon_Olcme_Aktif := "DB523.Pozisyon.Kontrol"."Pozisyon Olcme Aktif", Sağ_Çıkış_Target := 100, Sol_Çıkış_Target := 200, CN_NO := "DB531_FIFO_Kontrol".CN_NO[2].CNV_NO, "Aktüel Encoder Değeri" := "DB522.HSC".CN2.Encoder_Value_mm, Birinci_Divert_Min := "DB541_Divert_Control".Divert1_Min_Pos[1], Birinci_Divert_Max := "DB541_Divert_Control".Divert1_Max_Pos[1], İkinci_Divert_Min := "DB541_Divert_Control".Divert2_Min_Pos[1], İkinci_Divert_Max := "DB541_Divert_Control".Divert2_Max_Pos[1], Max_Kutu_Adedi := 10, "1_sol_Divert_Çalıştır" => "DB541_Divert_Control".SOL[1], "2_sol_Divert_Çalıştır" => "DB541_Divert_Control".SOl_2[1], "1_sağ_Divert_Çalıştır" => "DB541_Divert_Control".SAG[1], "2_sağ_Divert_Çalıştır" => "DB541_Divert_Control".SAG_2[1], "Sort Hatası" =>)
   END_RUNG
   RUNG wire#powerrail
      P_Contact(operand := "DB541_Divert_Control".SOL[1], bit := "AUX".BIT[58])
      { S7_Templates := "DestType := DInt" } Inc( "sayac" )
   END_RUNG
   // the same network as SCL:
   #Yanaştırma(Acil_Yok := #Acil_OK,   // "FB549.Divert.Sorter.Basing"
               Sorter_Calisiyor := #Otomatik,
               "Sağ_Chute_Aktif / Pasif" := true,
               "Sol_Chute_Aktif / Pasif" := true,
               Chute_Rulo_Hatası := false,
               Pozisyon_Olcme_Aktif := "DB523.Pozisyon.Kontrol"."Pozisyon Olcme Aktif",
               Sağ_Çıkış_Target := 100,
               Sol_Çıkış_Target := 200,
               CN_NO := "DB531_FIFO_Kontrol".CN_NO[2].CNV_NO,
               "Aktüel Encoder Değeri" := "DB522.HSC".CN2.Encoder_Value_mm,
               Birinci_Divert_Min := "DB541_Divert_Control".Divert1_Min_Pos[1],
               Birinci_Divert_Max := "DB541_Divert_Control".Divert1_Max_Pos[1],
               İkinci_Divert_Min := "DB541_Divert_Control".Divert2_Min_Pos[1],
               İkinci_Divert_Max := "DB541_Divert_Control".Divert2_Max_Pos[1],
               Max_Kutu_Adedi := 10,
               "1_sol_Divert_Çalıştır" => "DB541_Divert_Control".SOL[1],
               "2_sol_Divert_Çalıştır" => "DB541_Divert_Control".SOl_2[1],
               "1_sağ_Divert_Çalıştır" => "DB541_Divert_Control".SAG[1],
               "2_sağ_Divert_Çalıştır" => "DB541_Divert_Control".SAG_2[1]);
   #_w1 := "DB541_Divert_Control".SOL[1] AND NOT "AUX".BIT[58];   // rising edge of "DB541_Divert_Control".SOL[1]
   "AUX".BIT[58] := "DB541_Divert_Control".SOL[1];
   IF #_w1 THEN "sayac" := "sayac" + 1; END_IF;
END_REGION

REGION Network 2: CN3 POS1080 Divert2
   RUNG wire#powerrail
      #"FB548.Divert.Sorter.Chute_CN2_Divert2"(Acil_Yok := #Acil_OK, Sorter_Calisiyor := #Otomatik, Sağ_Chute_Sorted_Sensoru := "DB_ChuteSensors".DivertOut[1].Sorted.Sensor_N_Trig, Sol_Chute_Sorted_Sensoru := "DB_ChuteSensors".DivertOut[5].Sorted.Sensor_N_Trig, "Sağ_Chute_Aktif / Pasif" := true, "Sol_Chute_Aktif / Pasif" := true, Chute_Rulo_Hatası := false, Divert_Sürücü_Hatası :=, Pozisyon_Olcme_Aktif := "DB523.Pozisyon.Kontrol"."Pozisyon Olcme Aktif", Sağ_Çıkış_Target := 101, Sol_Çıkış_Target := 201, CN_NO := "DB531_FIFO_Kontrol".CN_NO[3].CNV_NO, "Aktüel Encoder Değeri" := "DB522.HSC".CN2.Encoder_Value_mm, Birinci_Divert_Min := "DB541_Divert_Control".Divert1_Min_Pos[2], Birinci_Divert_Max := "DB541_Divert_Control".Divert1_Max_Pos[2], İkinci_Divert_Min := "DB541_Divert_Control".Divert2_Min_Pos[2], İkinci_Divert_Max := "DB541_Divert_Control".Divert2_Max_Pos[2], Max_Kutu_Adedi := 10, "1_sol_Divert_Çalıştır" => "DB541_Divert_Control".SOL[2], "2_sol_Divert_Çalıştır" => "DB541_Divert_Control".SOl_2[2], "1_sağ_Divert_Çalıştır" => "DB541_Divert_Control".SAG[2], "2_sağ_Divert_Çalıştır" => "DB541_Divert_Control".SAG_2[2], "Sort Hatası" =>)
   END_RUNG
   // the same network as SCL:
   #"FB548.Divert.Sorter.Chute_CN2_Divert2"(Acil_Yok := #Acil_OK,   // "FB548.Divert.Sorter.Chute"
                           Sorter_Calisiyor := #Otomatik,
                           Sağ_Chute_Sorted_Sensoru := "DB_ChuteSensors".DivertOut[1].Sorted.Sensor_N_Trig,
                           Sol_Chute_Sorted_Sensoru := "DB_ChuteSensors".DivertOut[5].Sorted.Sensor_N_Trig,
                           "Sağ_Chute_Aktif / Pasif" := true,
                           "Sol_Chute_Aktif / Pasif" := true,
                           Chute_Rulo_Hatası := false,
                           Pozisyon_Olcme_Aktif := "DB523.Pozisyon.Kontrol"."Pozisyon Olcme Aktif",
                           Sağ_Çıkış_Target := 101,
                           Sol_Çıkış_Target := 201,
                           CN_NO := "DB531_FIFO_Kontrol".CN_NO[3].CNV_NO,
                           "Aktüel Encoder Değeri" := "DB522.HSC".CN2.Encoder_Value_mm,
                           Birinci_Divert_Min := "DB541_Divert_Control".Divert1_Min_Pos[2],
                           Birinci_Divert_Max := "DB541_Divert_Control".Divert1_Max_Pos[2],
                           İkinci_Divert_Min := "DB541_Divert_Control".Divert2_Min_Pos[2],
                           İkinci_Divert_Max := "DB541_Divert_Control".Divert2_Max_Pos[2],
                           Max_Kutu_Adedi := 10,
                           "1_sol_Divert_Çalıştır" => "DB541_Divert_Control".SOL[2],
                           "2_sol_Divert_Çalıştır" => "DB541_Divert_Control".SOl_2[2],
                           "1_sağ_Divert_Çalıştır" => "DB541_Divert_Control".SAG[2],
                           "2_sağ_Divert_Çalıştır" => "DB541_Divert_Control".SAG_2[2]);
END_REGION

REGION Network 3 (SCL)


   IF "DB541_Divert_Control".SOL[2] THEN
       "DB541_Divert_Control".SOl_2[2] := TRUE;
   END_IF;

   IF "DB541_Divert_Control".SAG[2] THEN
       "DB541_Divert_Control".SAG_2[2] := TRUE;
   END_IF;
END_REGION

REGION Network 4: CN4 POS1190 Divert3
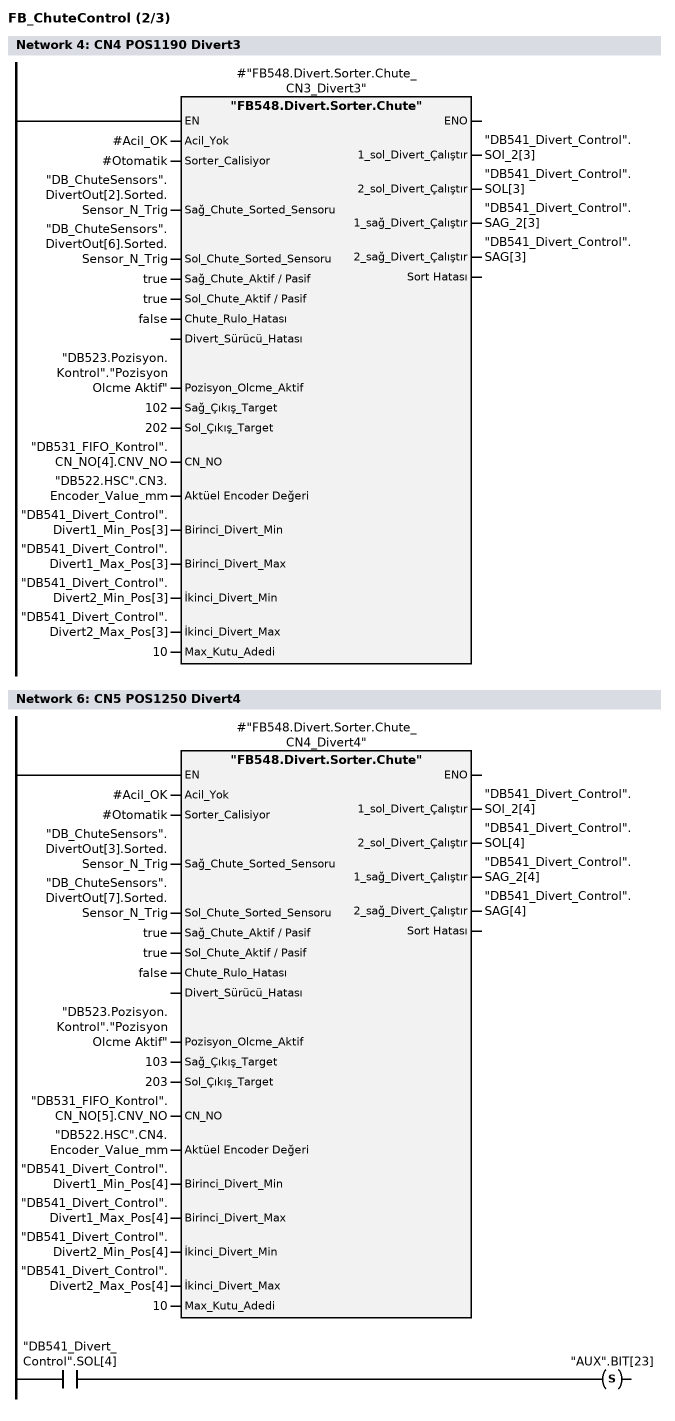
   RUNG wire#powerrail
      #"FB548.Divert.Sorter.Chute_CN3_Divert3"(Acil_Yok := #Acil_OK, Sorter_Calisiyor := #Otomatik, Sağ_Chute_Sorted_Sensoru := "DB_ChuteSensors".DivertOut[2].Sorted.Sensor_N_Trig, Sol_Chute_Sorted_Sensoru := "DB_ChuteSensors".DivertOut[6].Sorted.Sensor_N_Trig, "Sağ_Chute_Aktif / Pasif" := true, "Sol_Chute_Aktif / Pasif" := true, Chute_Rulo_Hatası := false, Divert_Sürücü_Hatası :=, Pozisyon_Olcme_Aktif := "DB523.Pozisyon.Kontrol"."Pozisyon Olcme Aktif", Sağ_Çıkış_Target := 102, Sol_Çıkış_Target := 202, CN_NO := "DB531_FIFO_Kontrol".CN_NO[4].CNV_NO, "Aktüel Encoder Değeri" := "DB522.HSC".CN3.Encoder_Value_mm, Birinci_Divert_Min := "DB541_Divert_Control".Divert1_Min_Pos[3], Birinci_Divert_Max := "DB541_Divert_Control".Divert1_Max_Pos[3], İkinci_Divert_Min := "DB541_Divert_Control".Divert2_Min_Pos[3], İkinci_Divert_Max := "DB541_Divert_Control".Divert2_Max_Pos[3], Max_Kutu_Adedi := 10, "1_sol_Divert_Çalıştır" => "DB541_Divert_Control".SOl_2[3], "2_sol_Divert_Çalıştır" => "DB541_Divert_Control".SOL[3], "1_sağ_Divert_Çalıştır" => "DB541_Divert_Control".SAG_2[3], "2_sağ_Divert_Çalıştır" => "DB541_Divert_Control".SAG[3], "Sort Hatası" =>)
   END_RUNG
   // the same network as SCL:
   #"FB548.Divert.Sorter.Chute_CN3_Divert3"(Acil_Yok := #Acil_OK,   // "FB548.Divert.Sorter.Chute"
                           Sorter_Calisiyor := #Otomatik,
                           Sağ_Chute_Sorted_Sensoru := "DB_ChuteSensors".DivertOut[2].Sorted.Sensor_N_Trig,
                           Sol_Chute_Sorted_Sensoru := "DB_ChuteSensors".DivertOut[6].Sorted.Sensor_N_Trig,
                           "Sağ_Chute_Aktif / Pasif" := true,
                           "Sol_Chute_Aktif / Pasif" := true,
                           Chute_Rulo_Hatası := false,
                           Pozisyon_Olcme_Aktif := "DB523.Pozisyon.Kontrol"."Pozisyon Olcme Aktif",
                           Sağ_Çıkış_Target := 102,
                           Sol_Çıkış_Target := 202,
                           CN_NO := "DB531_FIFO_Kontrol".CN_NO[4].CNV_NO,
                           "Aktüel Encoder Değeri" := "DB522.HSC".CN3.Encoder_Value_mm,
                           Birinci_Divert_Min := "DB541_Divert_Control".Divert1_Min_Pos[3],
                           Birinci_Divert_Max := "DB541_Divert_Control".Divert1_Max_Pos[3],
                           İkinci_Divert_Min := "DB541_Divert_Control".Divert2_Min_Pos[3],
                           İkinci_Divert_Max := "DB541_Divert_Control".Divert2_Max_Pos[3],
                           Max_Kutu_Adedi := 10,
                           "1_sol_Divert_Çalıştır" => "DB541_Divert_Control".SOl_2[3],
                           "2_sol_Divert_Çalıştır" => "DB541_Divert_Control".SOL[3],
                           "1_sağ_Divert_Çalıştır" => "DB541_Divert_Control".SAG_2[3],
                           "2_sağ_Divert_Çalıştır" => "DB541_Divert_Control".SAG[3]);
END_REGION

REGION Network 5 (SCL)


   IF "DB541_Divert_Control".SOl_2[3] THEN
       "DB541_Divert_Control".SOL[3] := TRUE;
   END_IF;

   IF "DB541_Divert_Control".SAG_2[3] THEN
       "DB541_Divert_Control".SAG[3] := TRUE;
   END_IF;
END_REGION

REGION Network 6: CN5 POS1250 Divert4
   RUNG wire#powerrail
      #"FB548.Divert.Sorter.Chute_CN4_Divert4"(Acil_Yok := #Acil_OK, Sorter_Calisiyor := #Otomatik, Sağ_Chute_Sorted_Sensoru := "DB_ChuteSensors".DivertOut[3].Sorted.Sensor_N_Trig, Sol_Chute_Sorted_Sensoru := "DB_ChuteSensors".DivertOut[7].Sorted.Sensor_N_Trig, "Sağ_Chute_Aktif / Pasif" := true, "Sol_Chute_Aktif / Pasif" := true, Chute_Rulo_Hatası := false, Divert_Sürücü_Hatası :=, Pozisyon_Olcme_Aktif := "DB523.Pozisyon.Kontrol"."Pozisyon Olcme Aktif", Sağ_Çıkış_Target := 103, Sol_Çıkış_Target := 203, CN_NO := "DB531_FIFO_Kontrol".CN_NO[5].CNV_NO, "Aktüel Encoder Değeri" := "DB522.HSC".CN4.Encoder_Value_mm, Birinci_Divert_Min := "DB541_Divert_Control".Divert1_Min_Pos[4], Birinci_Divert_Max := "DB541_Divert_Control".Divert1_Max_Pos[4], İkinci_Divert_Min := "DB541_Divert_Control".Divert2_Min_Pos[4], İkinci_Divert_Max := "DB541_Divert_Control".Divert2_Max_Pos[4], Max_Kutu_Adedi := 10, "1_sol_Divert_Çalıştır" => "DB541_Divert_Control".SOl_2[4], "2_sol_Divert_Çalıştır" => "DB541_Divert_Control".SOL[4], "1_sağ_Divert_Çalıştır" => "DB541_Divert_Control".SAG_2[4], "2_sağ_Divert_Çalıştır" => "DB541_Divert_Control".SAG[4], "Sort Hatası" =>)
   END_RUNG
   RUNG wire#powerrail
      Contact( "DB541_Divert_Control".SOL[4] )
      S_Coil( "AUX".BIT[23] )
   END_RUNG
   // the same network as SCL:
   #"FB548.Divert.Sorter.Chute_CN4_Divert4"(Acil_Yok := #Acil_OK,   // "FB548.Divert.Sorter.Chute"
                           Sorter_Calisiyor := #Otomatik,
                           Sağ_Chute_Sorted_Sensoru := "DB_ChuteSensors".DivertOut[3].Sorted.Sensor_N_Trig,
                           Sol_Chute_Sorted_Sensoru := "DB_ChuteSensors".DivertOut[7].Sorted.Sensor_N_Trig,
                           "Sağ_Chute_Aktif / Pasif" := true,
                           "Sol_Chute_Aktif / Pasif" := true,
                           Chute_Rulo_Hatası := false,
                           Pozisyon_Olcme_Aktif := "DB523.Pozisyon.Kontrol"."Pozisyon Olcme Aktif",
                           Sağ_Çıkış_Target := 103,
                           Sol_Çıkış_Target := 203,
                           CN_NO := "DB531_FIFO_Kontrol".CN_NO[5].CNV_NO,
                           "Aktüel Encoder Değeri" := "DB522.HSC".CN4.Encoder_Value_mm,
                           Birinci_Divert_Min := "DB541_Divert_Control".Divert1_Min_Pos[4],
                           Birinci_Divert_Max := "DB541_Divert_Control".Divert1_Max_Pos[4],
                           İkinci_Divert_Min := "DB541_Divert_Control".Divert2_Min_Pos[4],
                           İkinci_Divert_Max := "DB541_Divert_Control".Divert2_Max_Pos[4],
                           Max_Kutu_Adedi := 10,
                           "1_sol_Divert_Çalıştır" => "DB541_Divert_Control".SOl_2[4],
                           "2_sol_Divert_Çalıştır" => "DB541_Divert_Control".SOL[4],
                           "1_sağ_Divert_Çalıştır" => "DB541_Divert_Control".SAG_2[4],
                           "2_sağ_Divert_Çalıştır" => "DB541_Divert_Control".SAG[4]);
   IF "DB541_Divert_Control".SOL[4] THEN "AUX".BIT[23] := TRUE; END_IF;
END_REGION

REGION Network 7 (SCL)


   IF "DB541_Divert_Control".SOl_2[4] THEN
       "DB541_Divert_Control".SOL[4] := TRUE;
   END_IF;

   IF "DB541_Divert_Control".SAG_2[4] THEN
       "DB541_Divert_Control".SAG[4] := TRUE;
   END_IF;
END_REGION

REGION Network 8: CN6 POS1310 Divert5
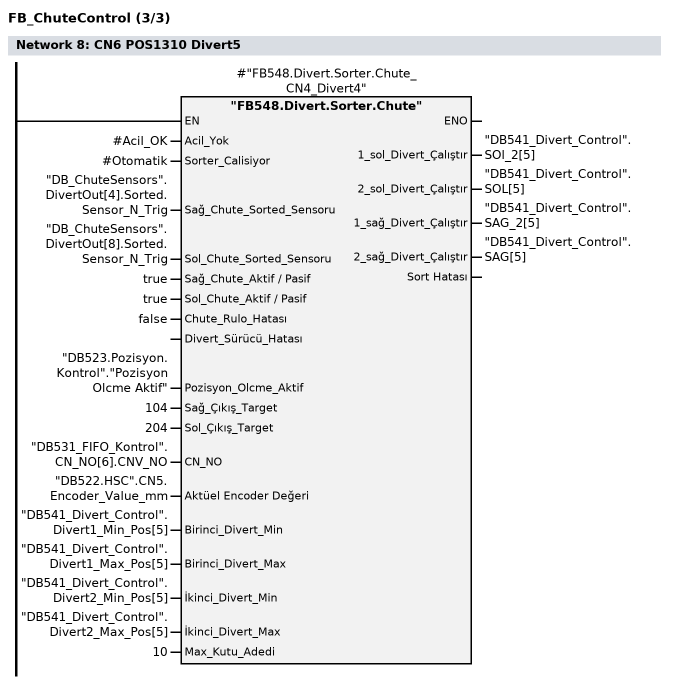
   RUNG wire#powerrail
      #"FB548.Divert.Sorter.Chute_CN4_Divert4"(Acil_Yok := #Acil_OK, Sorter_Calisiyor := #Otomatik, Sağ_Chute_Sorted_Sensoru := "DB_ChuteSensors".DivertOut[4].Sorted.Sensor_N_Trig, Sol_Chute_Sorted_Sensoru := "DB_ChuteSensors".DivertOut[8].Sorted.Sensor_N_Trig, "Sağ_Chute_Aktif / Pasif" := true, "Sol_Chute_Aktif / Pasif" := true, Chute_Rulo_Hatası := false, Divert_Sürücü_Hatası :=, Pozisyon_Olcme_Aktif := "DB523.Pozisyon.Kontrol"."Pozisyon Olcme Aktif", Sağ_Çıkış_Target := 104, Sol_Çıkış_Target := 204, CN_NO := "DB531_FIFO_Kontrol".CN_NO[6].CNV_NO, "Aktüel Encoder Değeri" := "DB522.HSC".CN5.Encoder_Value_mm, Birinci_Divert_Min := "DB541_Divert_Control".Divert1_Min_Pos[5], Birinci_Divert_Max := "DB541_Divert_Control".Divert1_Max_Pos[5], İkinci_Divert_Min := "DB541_Divert_Control".Divert2_Min_Pos[5], İkinci_Divert_Max := "DB541_Divert_Control".Divert2_Max_Pos[5], Max_Kutu_Adedi := 10, "1_sol_Divert_Çalıştır" => "DB541_Divert_Control".SOl_2[5], "2_sol_Divert_Çalıştır" => "DB541_Divert_Control".SOL[5], "1_sağ_Divert_Çalıştır" => "DB541_Divert_Control".SAG_2[5], "2_sağ_Divert_Çalıştır" => "DB541_Divert_Control".SAG[5], "Sort Hatası" =>)
   END_RUNG
   // the same network as SCL:
   #"FB548.Divert.Sorter.Chute_CN4_Divert4"(Acil_Yok := #Acil_OK,   // "FB548.Divert.Sorter.Chute"
                           Sorter_Calisiyor := #Otomatik,
                           Sağ_Chute_Sorted_Sensoru := "DB_ChuteSensors".DivertOut[4].Sorted.Sensor_N_Trig,
                           Sol_Chute_Sorted_Sensoru := "DB_ChuteSensors".DivertOut[8].Sorted.Sensor_N_Trig,
                           "Sağ_Chute_Aktif / Pasif" := true,
                           "Sol_Chute_Aktif / Pasif" := true,
                           Chute_Rulo_Hatası := false,
                           Pozisyon_Olcme_Aktif := "DB523.Pozisyon.Kontrol"."Pozisyon Olcme Aktif",
                           Sağ_Çıkış_Target := 104,
                           Sol_Çıkış_Target := 204,
                           CN_NO := "DB531_FIFO_Kontrol".CN_NO[6].CNV_NO,
                           "Aktüel Encoder Değeri" := "DB522.HSC".CN5.Encoder_Value_mm,
                           Birinci_Divert_Min := "DB541_Divert_Control".Divert1_Min_Pos[5],
                           Birinci_Divert_Max := "DB541_Divert_Control".Divert1_Max_Pos[5],
                           İkinci_Divert_Min := "DB541_Divert_Control".Divert2_Min_Pos[5],
                           İkinci_Divert_Max := "DB541_Divert_Control".Divert2_Max_Pos[5],
                           Max_Kutu_Adedi := 10,
                           "1_sol_Divert_Çalıştır" => "DB541_Divert_Control".SOl_2[5],
                           "2_sol_Divert_Çalıştır" => "DB541_Divert_Control".SOL[5],
                           "1_sağ_Divert_Çalıştır" => "DB541_Divert_Control".SAG_2[5],
                           "2_sağ_Divert_Çalıştır" => "DB541_Divert_Control".SAG[5]);
END_REGION

REGION Network 9 (SCL)


   IF "DB541_Divert_Control".SOl_2[5] THEN
       "DB541_Divert_Control".SOL[5] := TRUE;
   END_IF;

   IF "DB541_Divert_Control".SAG_2[5] THEN
       "DB541_Divert_Control".SAG[5] := TRUE;
   END_IF;
END_REGION
END_FUNCTION_BLOCK
